TYPE T_Ctrl_SIf_DPJ_DtChnToPLC :
STRUCT
	stNewDecision: T_Decision_DtChn;
END_STRUCT
END_TYPE

(* stored: Version 1.1.0.1, ProductVersion 3.1.0.19
   DUT T_Ctrl_SIf_DPJ_DtChnToPLC: Id {e1b6747f-c3c4-48e6-9fdf-2e87fe0093ca} *)
